Staubli VAL3: recvData.pgx

public program recvData(sio& x_sSioSocket, num& x_nRecvData[], RobotStatus& x_rRobotStatus, FlagStatus& x_fDataStatus, num& x_nRosFlagCmd)
  local num l_nRecvNum
begin

  //This program is used for receiving data from the host ROS controller.
  l_nRecvNum=sioGet(x_sSioSocket,x_nRecvData)
  if l_nRecvNum>0
    //call the decodeRecvData function to parse the received data
    call decodeRecvData(x_nRecvData,x_rRobotStatus,x_fDataStatus,x_nRosFlagCmd)
  endIf

end
